// TIA Portal V17 export
// export: Created 2023-04-11T09:33:28.3696619Z, ExportSetting WithDefaults, DisplayName Totally Integrated Automation Portal, DisplayVersion V17 Update 3, DisplayName TIA Portal Openness, DisplayVersion V17 Update 3, DisplayName TIA Portal Version Control Interface, DisplayVersion V17, DisplayName SINAMICS Startdrive Advanced, DisplayVersion V17 Update2, DisplayName SINAMICS Startdrive G130, G150, S120, S150, SINAMICS MV, S210, DisplayVersion V17 Update2, DisplayName SINAMICS Startdrive G110M, G120, G120C, G120D, G120P, G115D, DisplayVersion V17 Update2, DisplayName STEP 7 Professional, DisplayVersion V17 Update 3, DisplayName STEP 7 Safety, DisplayVersion V17, DisplayName WinCC UA Professional, DisplayVersion V17 Update 3
FUNCTION_BLOCK "StepBlock"   // FB20001, FBD
{ S7_Optimized_Access := 'TRUE' }
VERSION : 0.1
// stored: AutoNumber false, IsIECCheckEnabled false, IsRetainMemResEnabled false, MemoryReserve 100, SetENOAutomatically false, UDAEnableTagReadback false
   VAR_INPUT
      stepNumber : Int;
      activeStep : Int;
      conditions : Bool;
      delayCondition : Time;
      delayOutput : Time;
      delayAlarm : Time;
   END_VAR
   VAR_OUTPUT
      DONE : Bool;
      alarmBit : Bool;
      OUT_P : Bool;
      OUT : Bool;
      OUT_N : Bool;
   END_VAR
   VAR_IN_OUT
      index { ExternalAccessible := 'False'; ExternalVisible := 'False'; ExternalWritable := 'False'} : Int;
      HMI_text_tag : Array[0..2] of String;
      cnt : Int;   // counter for alarms and texts
   END_VAR
   VAR
      p_trig_1 : Bool;
      iec_timer_1 { S7_SetPoint := 'True'} : IEC_TIMER;
      iec_timer_2 { S7_SetPoint := 'True'} : IEC_TIMER;
      iec_timer_3 { S7_SetPoint := 'True'} : IEC_TIMER;
      edge_1 : Bool;
      edge_3 : Bool;
      enable { ExternalAccessible := 'False'; ExternalVisible := 'False'; ExternalWritable := 'False'} : Bool;
      edge_2 : Bool;
   END_VAR
   VAR_TEMP   // added for the SCL form of the ladder/FBD networks
      _w1 : Bool;
      _w2 : Bool;
   END_VAR
BEGIN

REGION Network 1: Enable Block
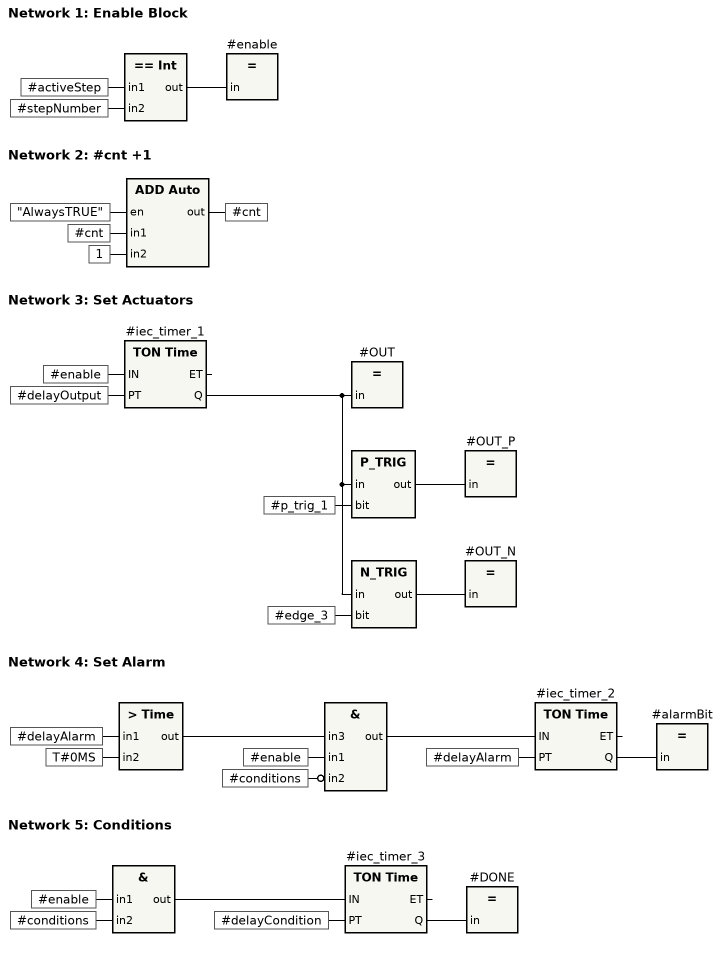
   #enable := #activeStep = #stepNumber;
END_REGION

REGION Network 2: #cnt +1
   IF "AlwaysTRUE" THEN #cnt := #cnt + 1; END_IF;
END_REGION

REGION Network 3: Set Actuators
   // Actuator_S - Set output as long as step is active
   // Actuator_P - Pulse output
   #iec_timer_1.TON(IN := #enable, PT := #delayOutput);
   #OUT := #iec_timer_1.Q;
   #_w1 := #iec_timer_1.Q AND NOT #p_trig_1;   // rising edge
   #p_trig_1 := #iec_timer_1.Q;
   #OUT_P := #_w1;
   #_w2 := NOT #iec_timer_1.Q AND #edge_3;   // falling edge
   #edge_3 := #iec_timer_1.Q;
   #OUT_N := #_w2;
END_REGION

REGION Network 4: Set Alarm
   #iec_timer_2.TON(IN := (#delayAlarm > T#0MS) AND #enable AND NOT #conditions, PT := #delayAlarm);
   #alarmBit := #iec_timer_2.Q;
END_REGION

REGION Network 5: Conditions
   // Step conditions to proceed to next step
   #iec_timer_3.TON(IN := #enable AND #conditions, PT := #delayCondition);
   #DONE := #iec_timer_3.Q;
END_REGION
END_FUNCTION_BLOCK
